# EPICS autosave request: recipes-examples/demo-ioc/files/iocBoot/iocdemo/auto.req
# SPDX-FileCopyrightText: 2026 IMPCAS
#
# SPDX-License-Identifier: MIT

# Records saved by autosave. $(P) is supplied when the set is created.

$(P)cmdset
$(P)cmd
